Staubli VAL3: onF2Event.pgx

program onF2Event(bool& x_bSave[] (dimensions=1))
  local string l_sPath
  local string l_sItems[2]
begin
  // look if the bButton is enable
  if bButton[1]
    //
    // edit all the pallet point
    //
    if x_bSave
      // saver IT
      call saveIt(x_bSave)
    endIf
    // load the page viewTraj
    l_sPath="Disk://trajectory/page_viewTraj"
    l_sItems=sPalletName
    nPosition=nPosition-1
    l_sItems[1]=toString("",max(nPosition[0],0))
    call loadPage(l_sPath,l_sItems)
    // came back
    if l_sItems[0]=="saved"
      x_bSave=false
    endIf
    //
    call buildList()
    //
  endIf
end
